// SIMATIC S7-200 SMART project (STEP 7-Micro/WIN SMART), CPU ST20

SYMBOL_TABLE 系统符号
Always_On        SM0.0    // 始终接通
First_Scan_On    SM0.1    // 仅在第一个扫描周期时接通
Clock_1s         SM0.5    // 针对 1 s 的周期时间，时钟脉冲接通 0.5 s，断开 0.5 s.
Time_0_Intrvl    SMB34    // 指定中断 0 的时间间隔（从 5 到 255，以 1 毫秒递增）。
END_SYMBOL_TABLE

ORGANIZATION_BLOCK MAIN:OB1
TITLE=程序注释
BEGIN
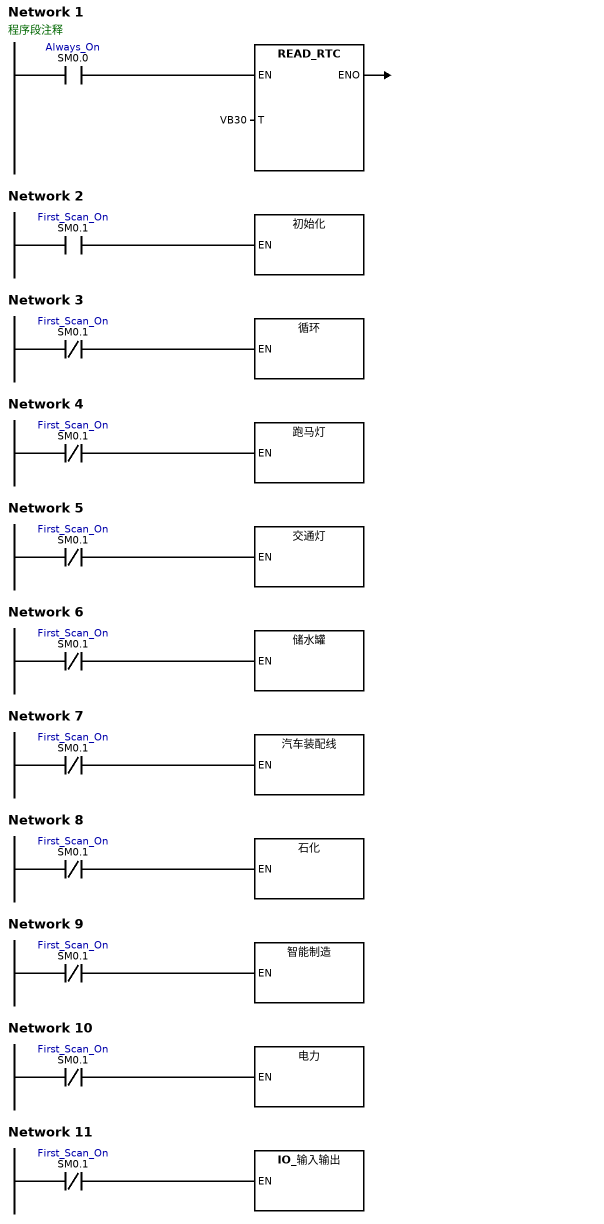
Network 1
// 程序段注释
LD     Always_On:SM0.0
TODR   VB30
Network 2
LD     First_Scan_On:SM0.1
CALL   初始化:SBR4
Network 3
LDN    First_Scan_On:SM0.1
CALL   循环:SBR14
Network 4
LDN    First_Scan_On:SM0.1
CALL   跑马灯:SBR0
Network 5
LDN    First_Scan_On:SM0.1
CALL   交通灯:SBR2
Network 6
// (network saved uncompiled; LAD cells follow)
// row 0: c0 -|/|- First_Scan_On:SM0.1  c1 --  c2 [储水罐 EN:=power@row0]
Network 7
LDN    First_Scan_On:SM0.1
CALL   汽车装配线:SBR7
Network 8
LDN    First_Scan_On:SM0.1
CALL   石化:SBR8
Network 9
LDN    First_Scan_On:SM0.1
CALL   智能制造:SBR9
Network 10
LDN    First_Scan_On:SM0.1
CALL   电力:SBR11
Network 11
LDN    First_Scan_On:SM0.1
CALL   IO_输入输出:SBR13
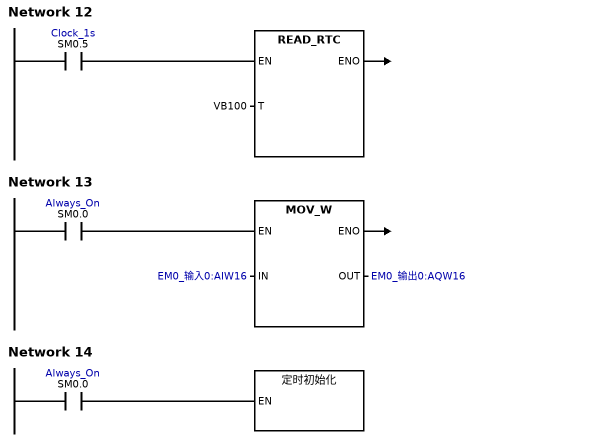
Network 12
LD     Clock_1s:SM0.5
TODR   VB100
Network 13
LD     Always_On:SM0.0
MOVW   EM0_输入0:AIW16, EM0_输出0:AQW16
Network 14
LD     Always_On:SM0.0
CALL   定时初始化:SBR1
END_ORGANIZATION_BLOCK

SUBROUTINE_BLOCK 跑马灯:SBR0
TITLE=子程序注释
BEGIN
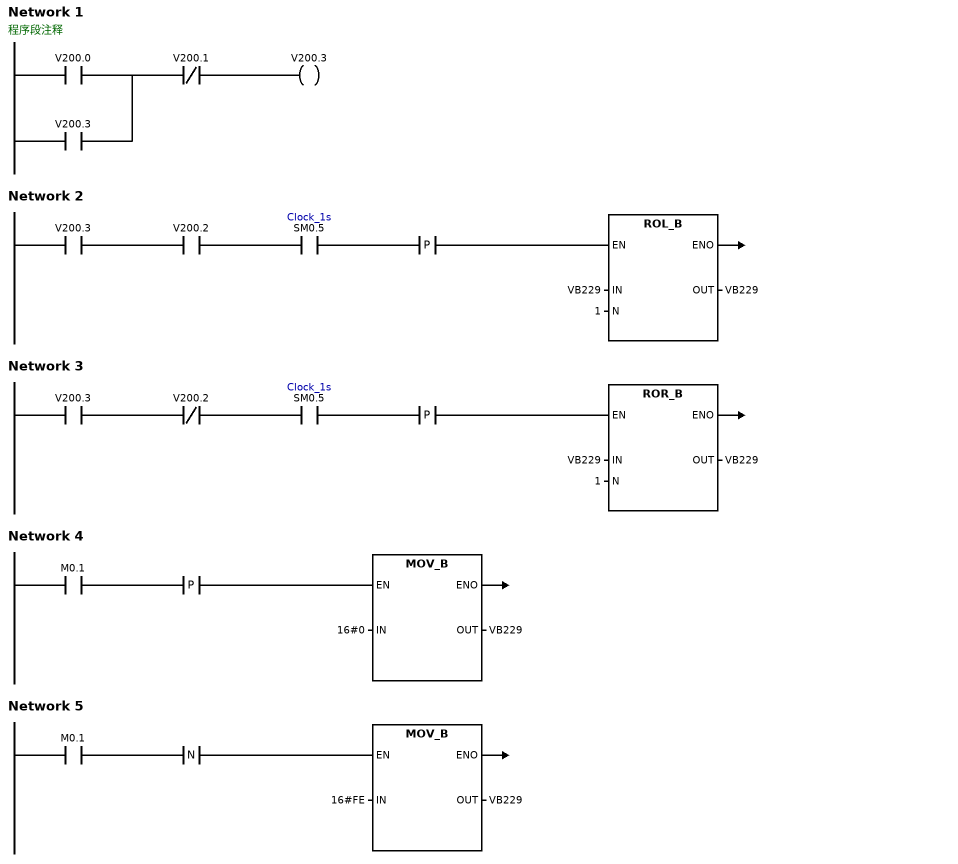
Network 1
// 程序段注释
LD     V200.0
O      V200.3
AN     V200.1
=      V200.3
Network 2
LD     V200.3
A      V200.2
A      Clock_1s:SM0.5
EU
RLB    VB229, 1
Network 3
LD     V200.3
AN     V200.2
A      Clock_1s:SM0.5
EU
RRB    VB229, 1
Network 4
LD     M0.1
EU
MOVB   16#0, VB229
Network 5
LD     M0.1
ED
MOVB   16#FE, VB229
END_SUBROUTINE_BLOCK

SUBROUTINE_BLOCK 定时初始化:SBR1
TITLE=
BEGIN
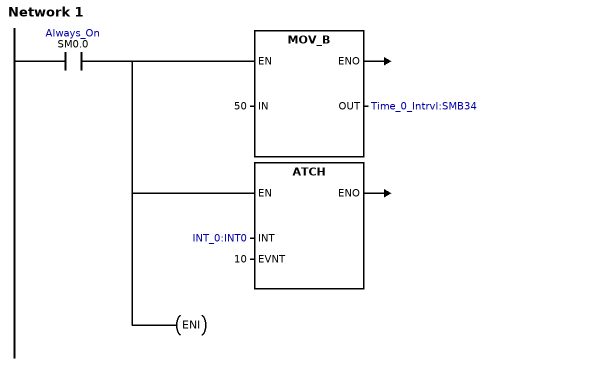
Network 1
LD     Always_On:SM0.0
MOVB   50, Time_0_Intrvl:SMB34
ATCH   INT_0:INT0, 10
ENI
END_SUBROUTINE_BLOCK

SUBROUTINE_BLOCK 交通灯:SBR2
TITLE=
BEGIN
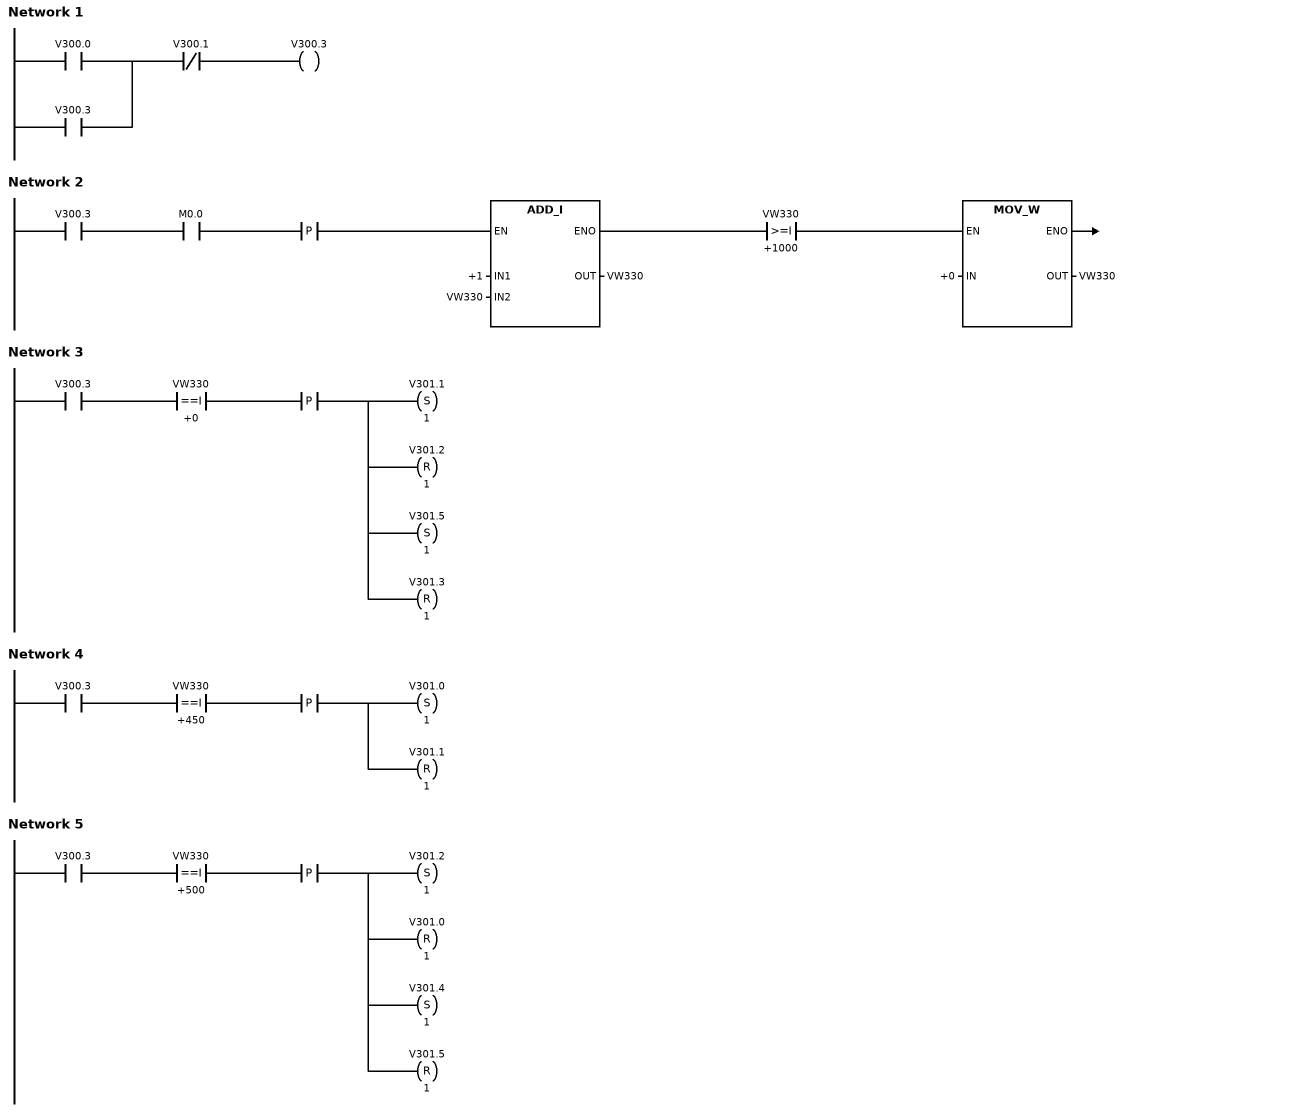
Network 1
LD     V300.0
O      V300.3
AN     V300.1
=      V300.3
Network 2
LD     V300.3
A      M0.0
EU
+I     +1, VW330
AENO
AW>=   VW330, +1000
MOVW   +0, VW330
Network 3
LD     V300.3
AW=    VW330, +0
EU
S      V301.1, 1
R      V301.2, 1
S      V301.5, 1
R      V301.3, 1
Network 4
LD     V300.3
AW=    VW330, +450
EU
S      V301.0, 1
R      V301.1, 1
Network 5
LD     V300.3
AW=    VW330, +500
EU
S      V301.2, 1
R      V301.0, 1
S      V301.4, 1
R      V301.5, 1
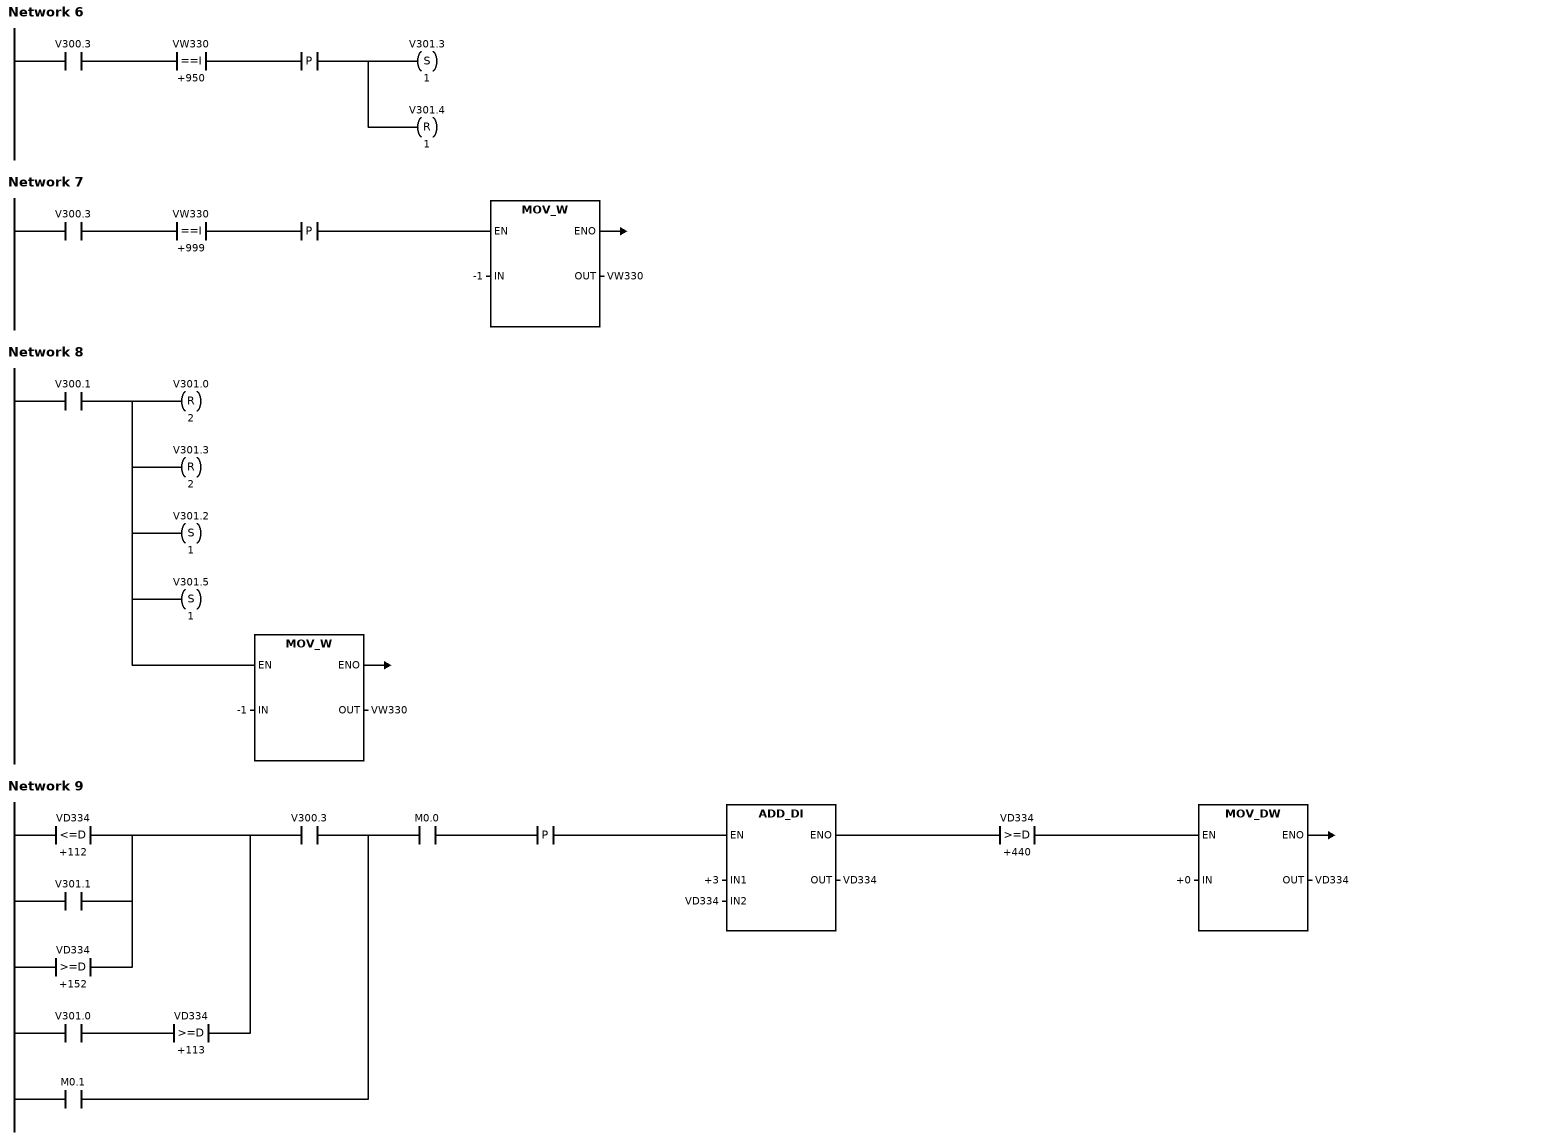
Network 6
LD     V300.3
AW=    VW330, +950
EU
S      V301.3, 1
R      V301.4, 1
Network 7
LD     V300.3
AW=    VW330, +999
EU
MOVW   -1, VW330
Network 8
LD     V300.1
R      V301.0, 2
R      V301.3, 2
S      V301.2, 1
S      V301.5, 1
MOVW   -1, VW330
Network 9
LDD<=  VD334, +112
O      V301.1
OD>=   VD334, +152
LD     V301.0
AD>=   VD334, +113
OLD
A      V300.3
O      M0.1
A      M0.0
EU
+D     +3, VD334
AENO
AD>=   VD334, +440
MOVD   +0, VD334
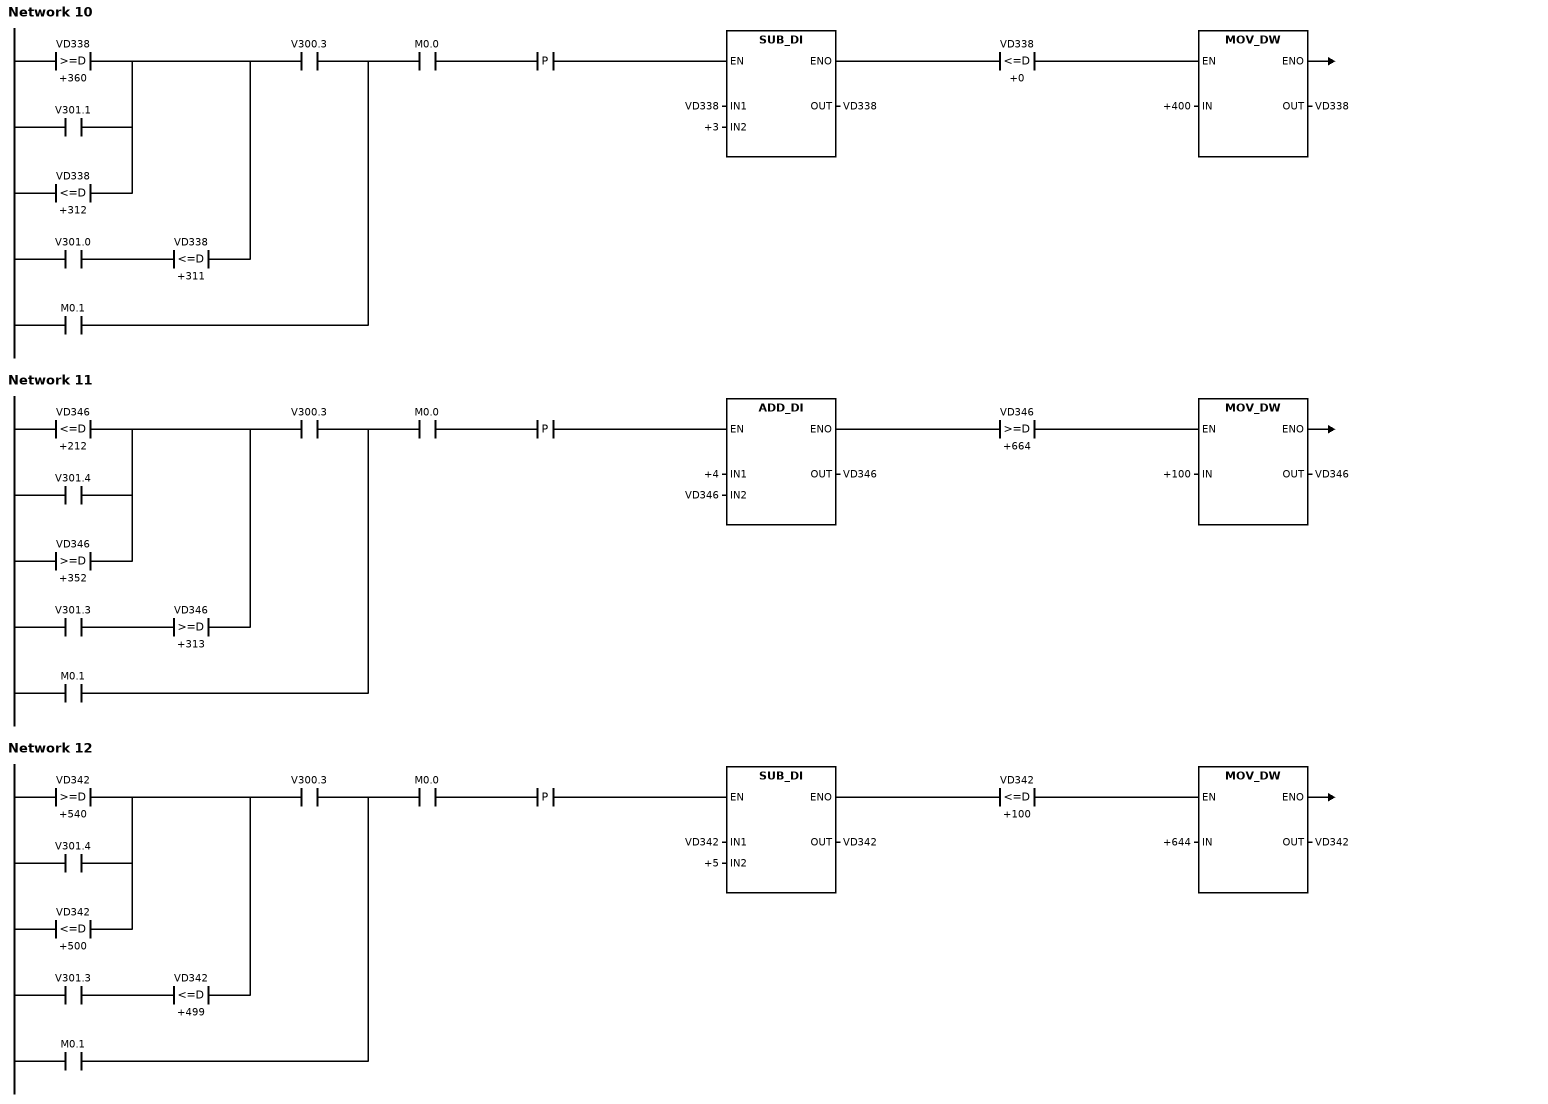
Network 10
LDD>=  VD338, +360
O      V301.1
OD<=   VD338, +312
LD     V301.0
AD<=   VD338, +311
OLD
A      V300.3
O      M0.1
A      M0.0
EU
-D     +3, VD338
AENO
AD<=   VD338, +0
MOVD   +400, VD338
Network 11
LDD<=  VD346, +212
O      V301.4
OD>=   VD346, +352
LD     V301.3
AD>=   VD346, +313
OLD
A      V300.3
O      M0.1
A      M0.0
EU
+D     +4, VD346
AENO
AD>=   VD346, +664
MOVD   +100, VD346
Network 12
LDD>=  VD342, +540
O      V301.4
OD<=   VD342, +500
LD     V301.3
AD<=   VD342, +499
OLD
A      V300.3
O      M0.1
A      M0.0
EU
-D     +5, VD342
AENO
AD<=   VD342, +100
MOVD   +644, VD342
END_SUBROUTINE_BLOCK

SUBROUTINE_BLOCK 模拟量输出:SBR3
TITLE=
VAR_INPUT
In_Data:REAL;	// LD0 
HH:REAL;	// LD4 
LL:REAL;	// LD8 
END_VAR
VAR_OUTPUT
AQW_:INT;	// LW12 
END_VAR
BEGIN
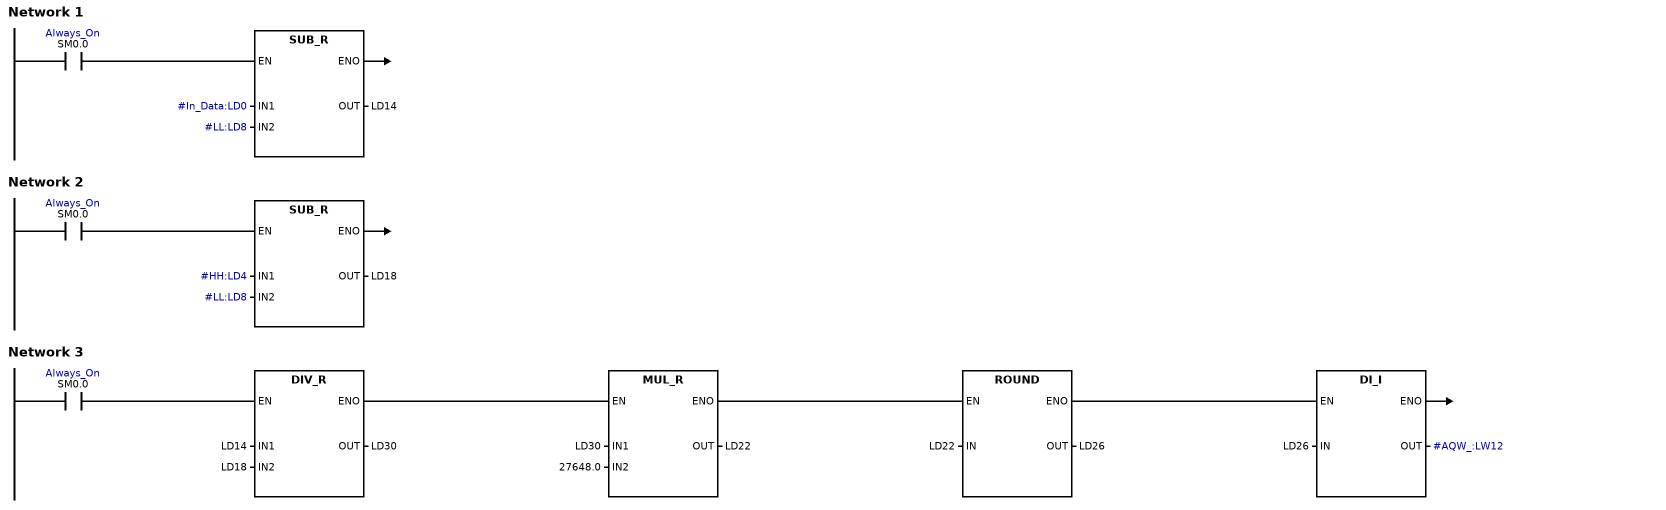
Network 1
LD     Always_On:SM0.0
MOVR   #In_Data:LD0, LD14
-R     #LL:LD8, LD14
Network 2
LD     Always_On:SM0.0
MOVR   #HH:LD4, LD18
-R     #LL:LD8, LD18
Network 3
LD     Always_On:SM0.0
MOVR   LD14, LD30
AENO
/R     LD18, LD30
AENO
MOVR   LD30, LD22
AENO
*R     27648.0, LD22
AENO
ROUND  LD22, LD26
AENO
DTI    LD26, #AQW_:LW12
END_SUBROUTINE_BLOCK

SUBROUTINE_BLOCK 初始化:SBR4
TITLE=
BEGIN
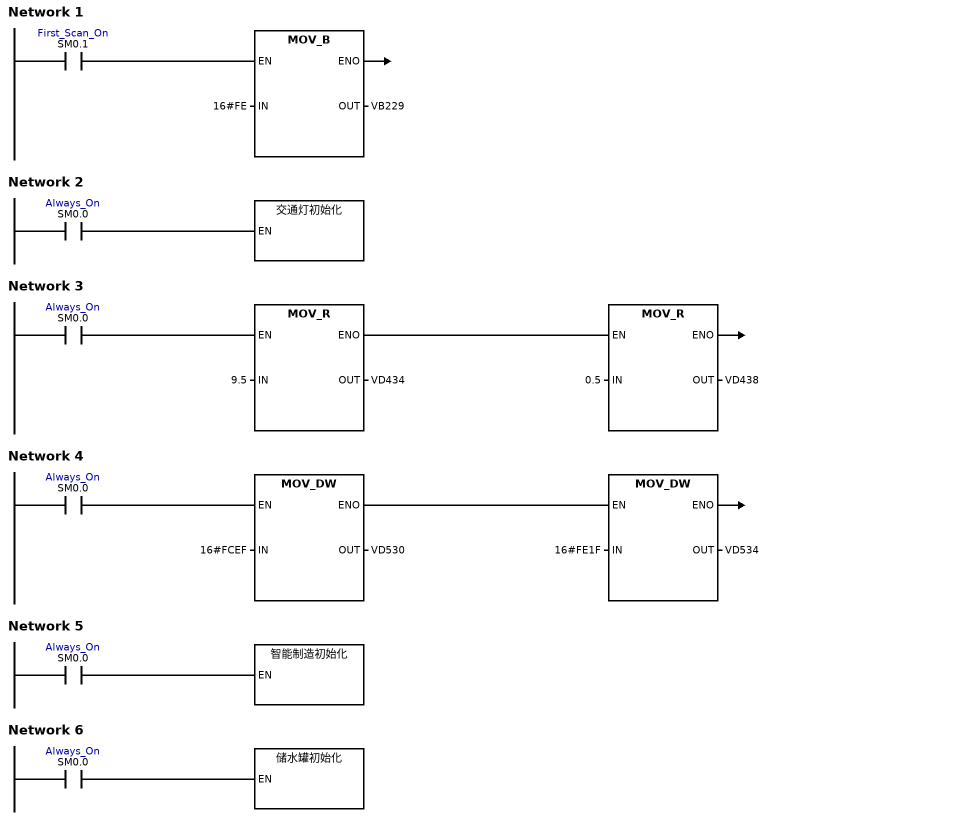
Network 1
LD     First_Scan_On:SM0.1
MOVB   16#FE, VB229
Network 2
LD     Always_On:SM0.0
CALL   交通灯初始化:SBR5
Network 3
LD     Always_On:SM0.0
MOVR   9.5, VD434
AENO
MOVR   0.5, VD438
Network 4
LD     Always_On:SM0.0
MOVD   16#FCEF, VD530
AENO
MOVD   16#FE1F, VD534
Network 5
LD     Always_On:SM0.0
CALL   智能制造初始化:SBR10
Network 6
LD     Always_On:SM0.0
CALL   储水罐初始化:SBR12
END_SUBROUTINE_BLOCK

SUBROUTINE_BLOCK 交通灯初始化:SBR5
TITLE=
BEGIN
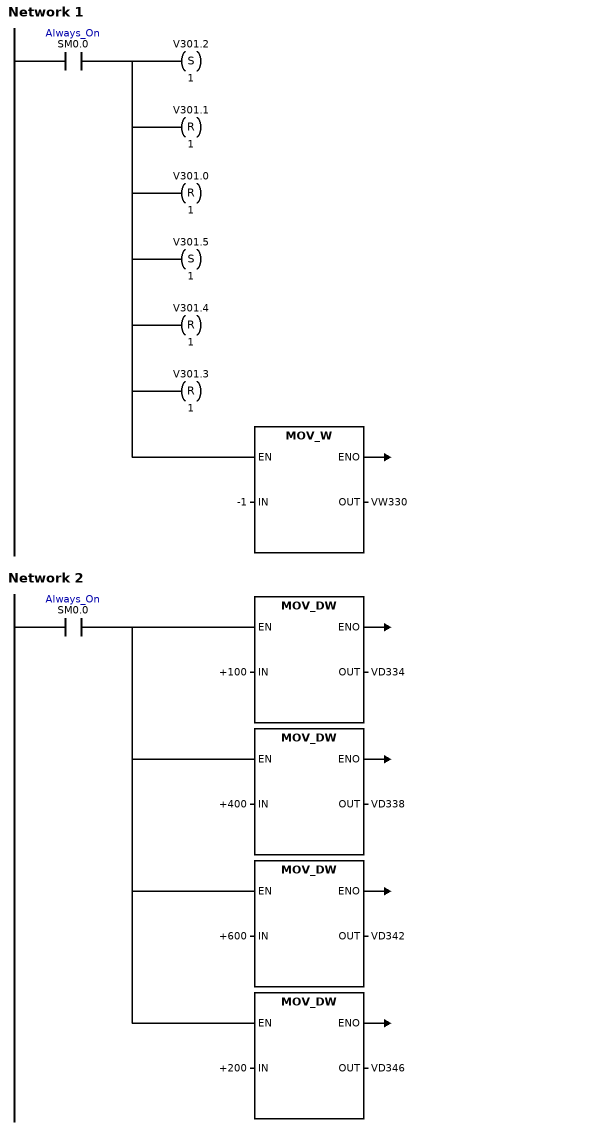
Network 1
LD     Always_On:SM0.0
S      V301.2, 1
R      V301.1, 1
R      V301.0, 1
S      V301.5, 1
R      V301.4, 1
R      V301.3, 1
MOVW   -1, VW330
Network 2
LD     Always_On:SM0.0
MOVD   +100, VD334
MOVD   +400, VD338
MOVD   +600, VD342
MOVD   +200, VD346
END_SUBROUTINE_BLOCK

SUBROUTINE_BLOCK 储水罐:SBR6
TITLE=
BEGIN
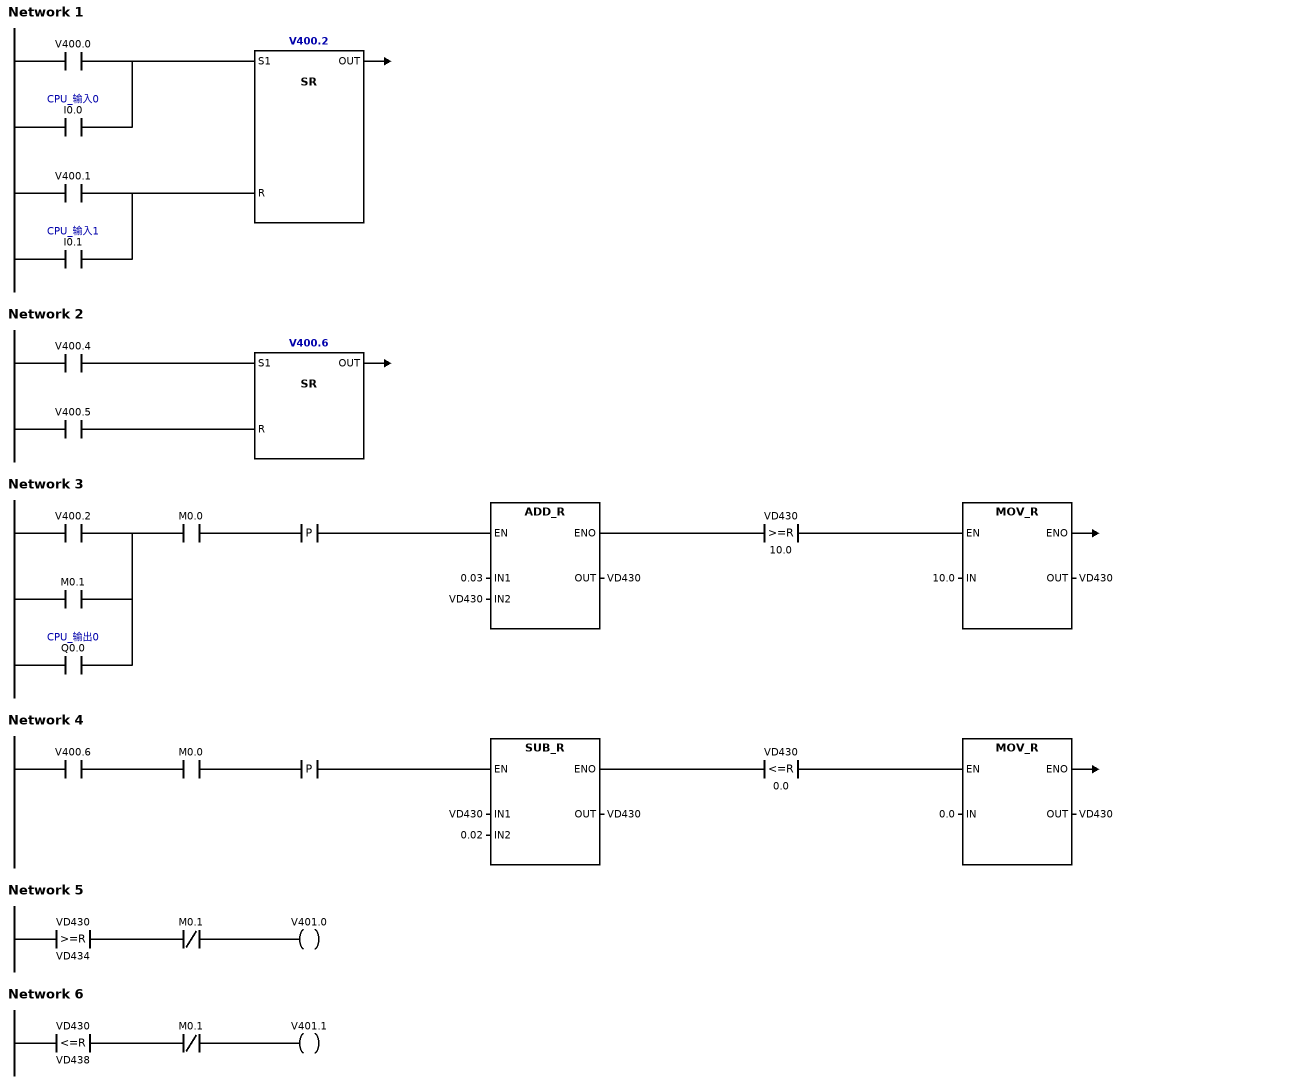
Network 1
LD     V400.0
O      CPU_输入0:I0.0
LD     V400.1
O      CPU_输入1:I0.1
NOT
A      V400.2
OLD
=      V400.2
Network 2
LD     V400.4
LD     V400.5
NOT
A      V400.6
OLD
=      V400.6
Network 3
LD     V400.2
O      M0.1
O      CPU_输出0:Q0.0
A      M0.0
EU
+R     0.03, VD430
AENO
AR>=   VD430, 10.0
MOVR   10.0, VD430
Network 4
LD     V400.6
A      M0.0
EU
-R     0.02, VD430
AENO
AR<=   VD430, 0.0
MOVR   0.0, VD430
Network 5
LDR>=  VD430, VD434
AN     M0.1
=      V401.0
Network 6
LDR<=  VD430, VD438
AN     M0.1
=      V401.1
END_SUBROUTINE_BLOCK

SUBROUTINE_BLOCK 汽车装配线:SBR7
TITLE=
BEGIN
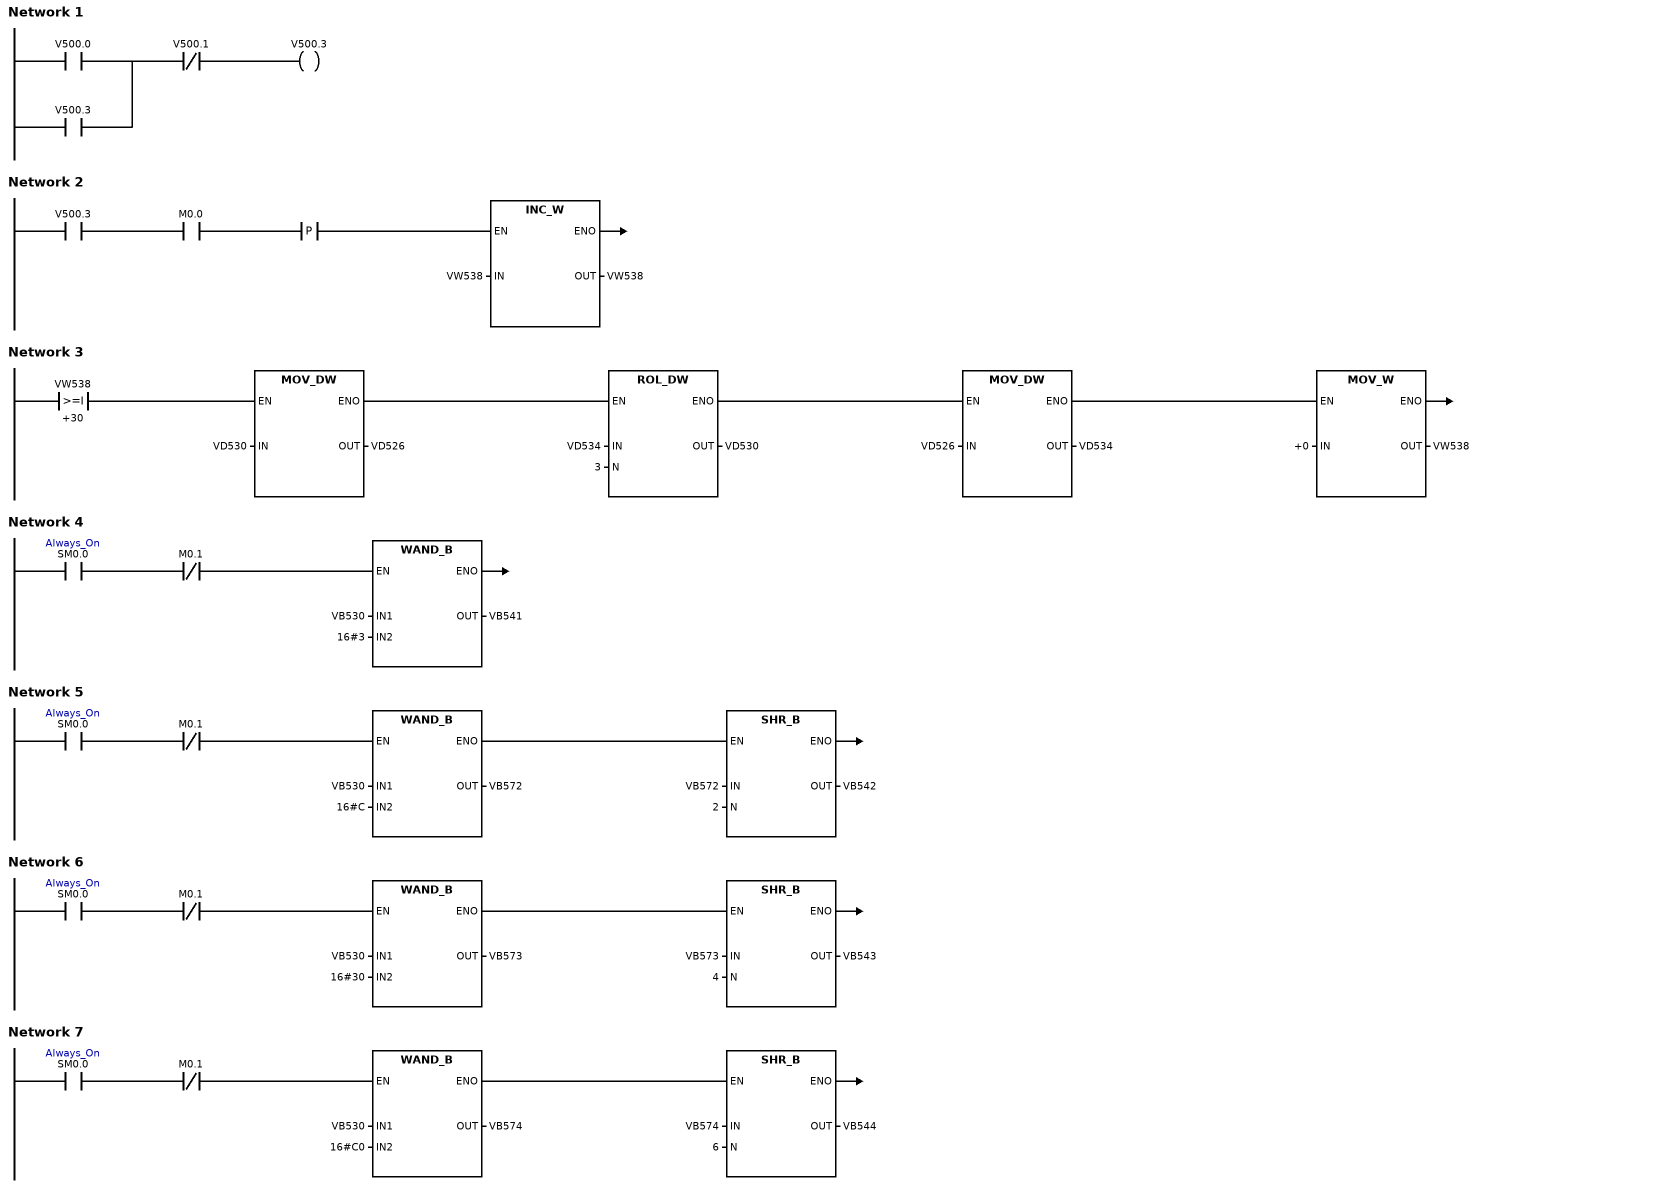
Network 1
LD     V500.0
O      V500.3
AN     V500.1
=      V500.3
Network 2
LD     V500.3
A      M0.0
EU
INCW   VW538
Network 3
LDW>=  VW538, +30
MOVD   VD530, VD526
AENO
MOVD   VD534, VD530
AENO
RLD    VD530, 3
AENO
MOVD   VD526, VD534
AENO
MOVW   +0, VW538
Network 4
LD     Always_On:SM0.0
AN     M0.1
MOVB   VB530, VB541
ANDB   16#3, VB541
Network 5
LD     Always_On:SM0.0
AN     M0.1
MOVB   VB530, VB572
AENO
ANDB   16#C, VB572
AENO
MOVB   VB572, VB542
SRB    VB542, 2
Network 6
LD     Always_On:SM0.0
AN     M0.1
MOVB   VB530, VB573
AENO
ANDB   16#30, VB573
AENO
MOVB   VB573, VB543
SRB    VB543, 4
Network 7
LD     Always_On:SM0.0
AN     M0.1
MOVB   VB530, VB574
AENO
ANDB   16#C0, VB574
AENO
MOVB   VB574, VB544
SRB    VB544, 6
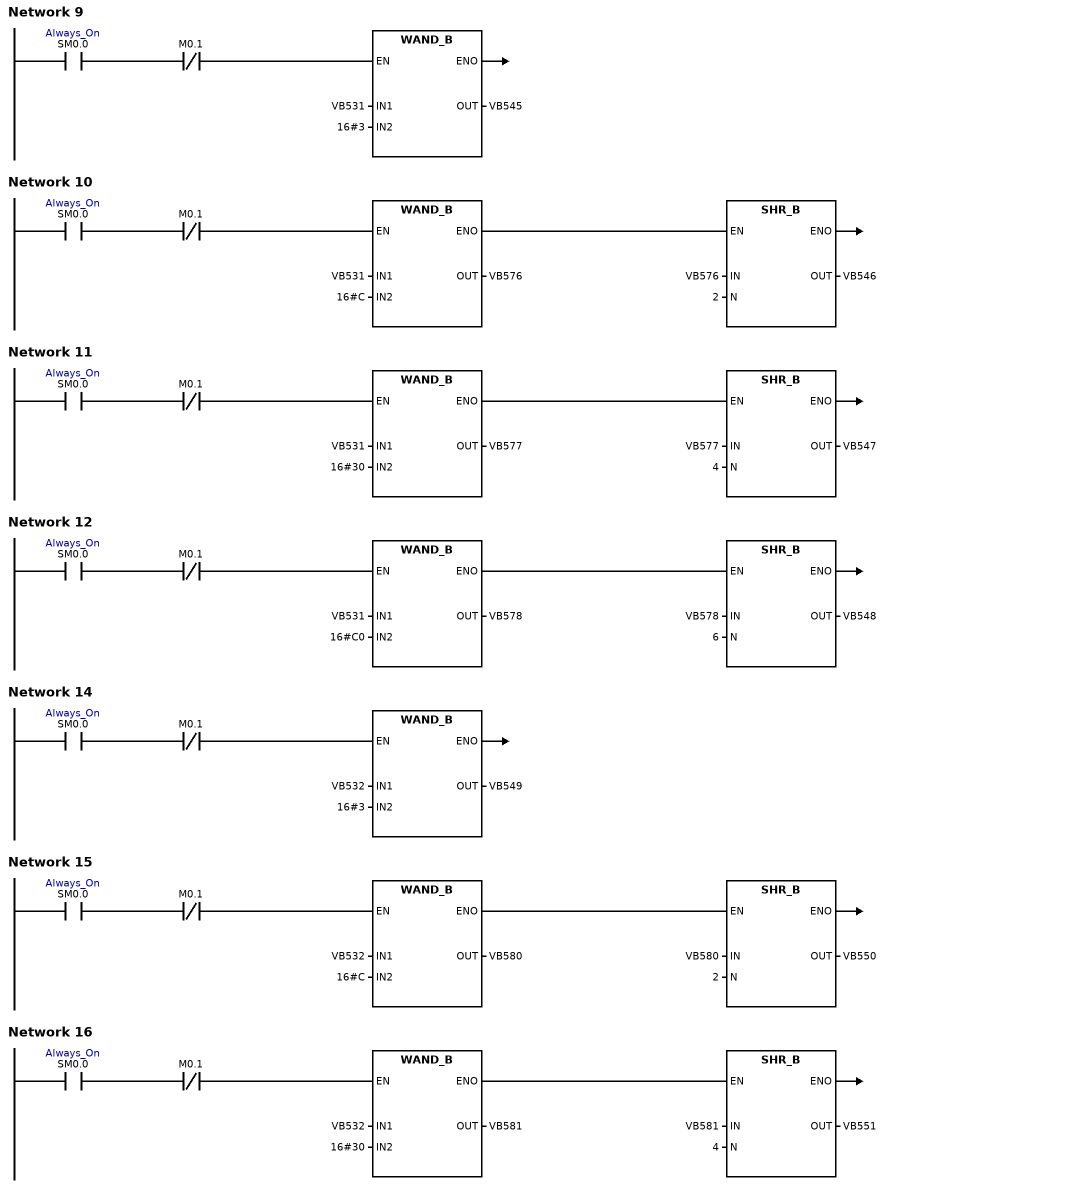
Network 9
LD     Always_On:SM0.0
AN     M0.1
MOVB   VB531, VB545
ANDB   16#3, VB545
Network 10
LD     Always_On:SM0.0
AN     M0.1
MOVB   VB531, VB576
AENO
ANDB   16#C, VB576
AENO
MOVB   VB576, VB546
SRB    VB546, 2
Network 11
LD     Always_On:SM0.0
AN     M0.1
MOVB   VB531, VB577
AENO
ANDB   16#30, VB577
AENO
MOVB   VB577, VB547
SRB    VB547, 4
Network 12
LD     Always_On:SM0.0
AN     M0.1
MOVB   VB531, VB578
AENO
ANDB   16#C0, VB578
AENO
MOVB   VB578, VB548
SRB    VB548, 6
Network 14
LD     Always_On:SM0.0
AN     M0.1
MOVB   VB532, VB549
ANDB   16#3, VB549
Network 15
LD     Always_On:SM0.0
AN     M0.1
MOVB   VB532, VB580
AENO
ANDB   16#C, VB580
AENO
MOVB   VB580, VB550
SRB    VB550, 2
Network 16
LD     Always_On:SM0.0
AN     M0.1
MOVB   VB532, VB581
AENO
ANDB   16#30, VB581
AENO
MOVB   VB581, VB551
SRB    VB551, 4
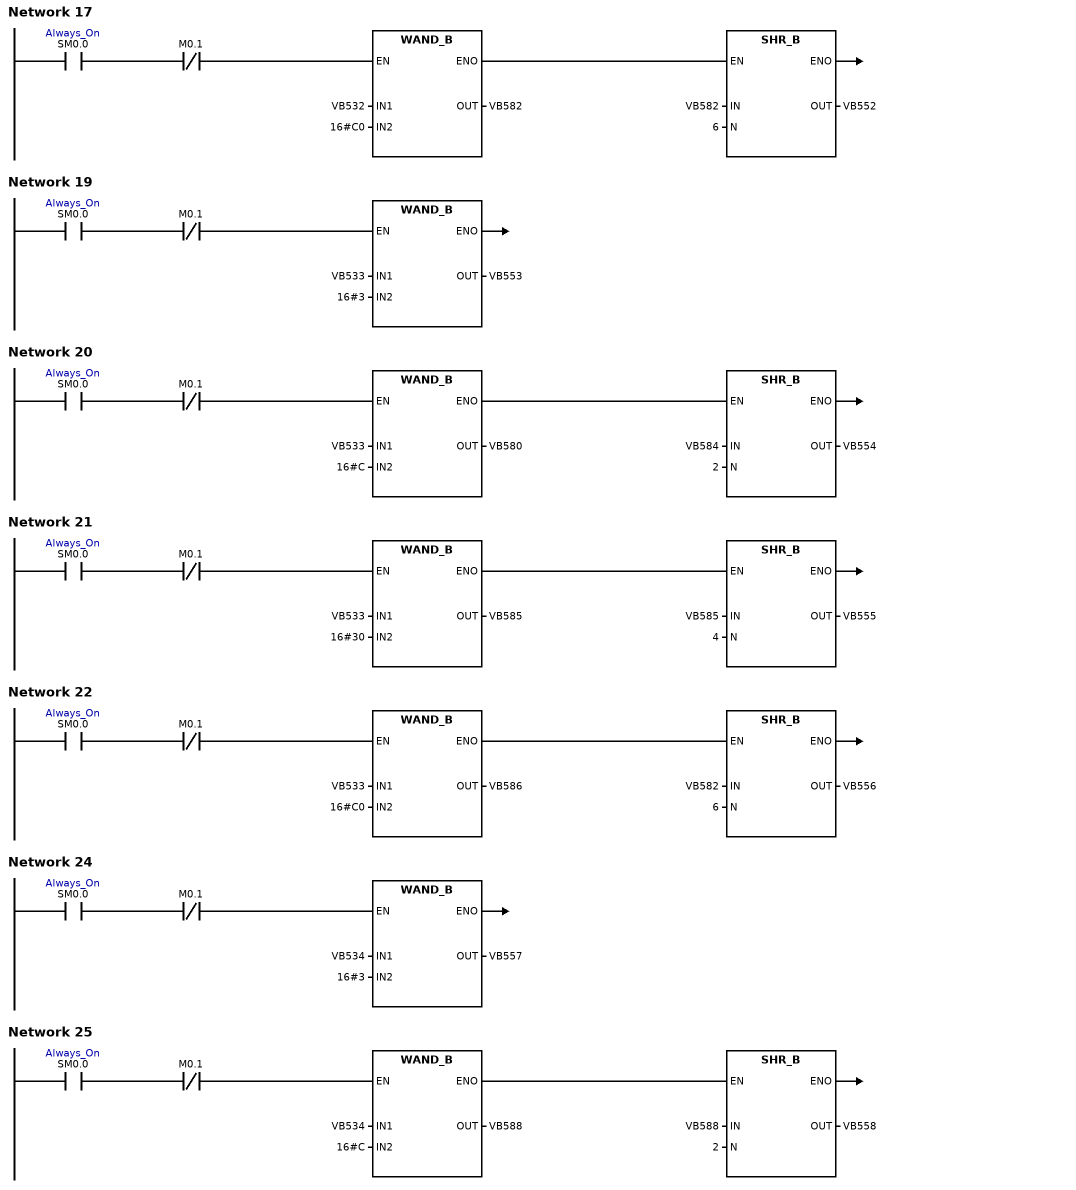
Network 17
LD     Always_On:SM0.0
AN     M0.1
MOVB   VB532, VB582
AENO
ANDB   16#C0, VB582
AENO
MOVB   VB582, VB552
SRB    VB552, 6
Network 19
LD     Always_On:SM0.0
AN     M0.1
MOVB   VB533, VB553
ANDB   16#3, VB553
Network 20
LD     Always_On:SM0.0
AN     M0.1
MOVB   VB533, VB580
AENO
ANDB   16#C, VB580
AENO
MOVB   VB584, VB554
SRB    VB554, 2
Network 21
LD     Always_On:SM0.0
AN     M0.1
MOVB   VB533, VB585
AENO
ANDB   16#30, VB585
AENO
MOVB   VB585, VB555
SRB    VB555, 4
Network 22
LD     Always_On:SM0.0
AN     M0.1
MOVB   VB533, VB586
AENO
ANDB   16#C0, VB586
AENO
MOVB   VB582, VB556
SRB    VB556, 6
Network 24
LD     Always_On:SM0.0
AN     M0.1
MOVB   VB534, VB557
ANDB   16#3, VB557
Network 25
LD     Always_On:SM0.0
AN     M0.1
MOVB   VB534, VB588
AENO
ANDB   16#C, VB588
AENO
MOVB   VB588, VB558
SRB    VB558, 2
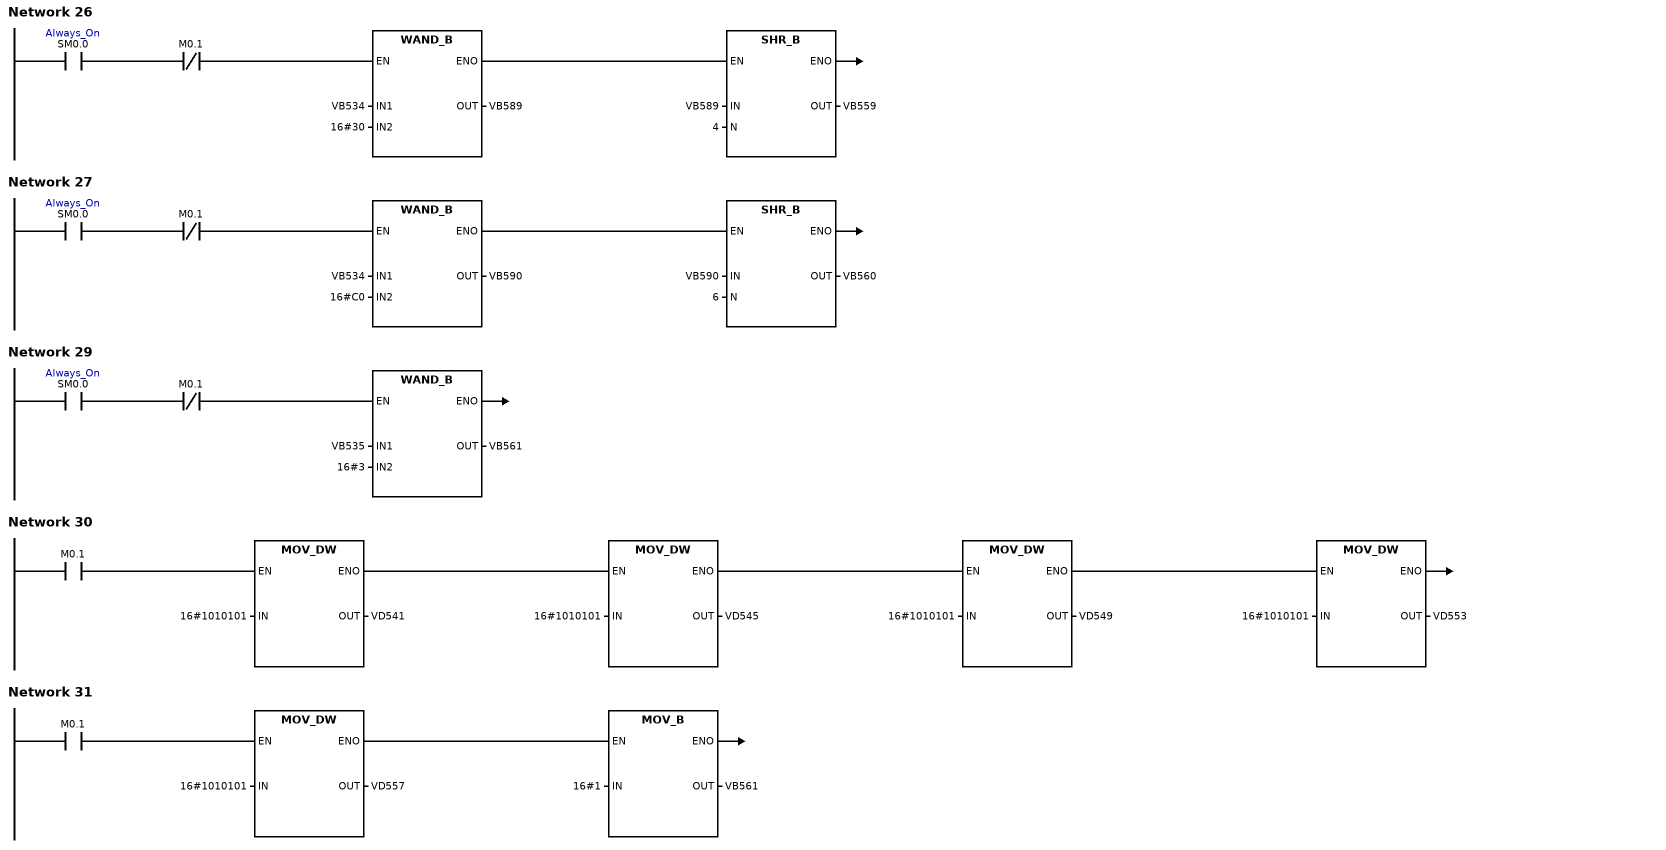
Network 26
LD     Always_On:SM0.0
AN     M0.1
MOVB   VB534, VB589
AENO
ANDB   16#30, VB589
AENO
MOVB   VB589, VB559
SRB    VB559, 4
Network 27
LD     Always_On:SM0.0
AN     M0.1
MOVB   VB534, VB590
AENO
ANDB   16#C0, VB590
AENO
MOVB   VB590, VB560
SRB    VB560, 6
Network 29
LD     Always_On:SM0.0
AN     M0.1
MOVB   VB535, VB561
ANDB   16#3, VB561
Network 30
LD     M0.1
MOVD   16#1010101, VD541
AENO
MOVD   16#1010101, VD545
AENO
MOVD   16#1010101, VD549
AENO
MOVD   16#1010101, VD553
Network 31
LD     M0.1
MOVD   16#1010101, VD557
AENO
MOVB   16#1, VB561
END_SUBROUTINE_BLOCK

SUBROUTINE_BLOCK 石化:SBR8
TITLE=
BEGIN
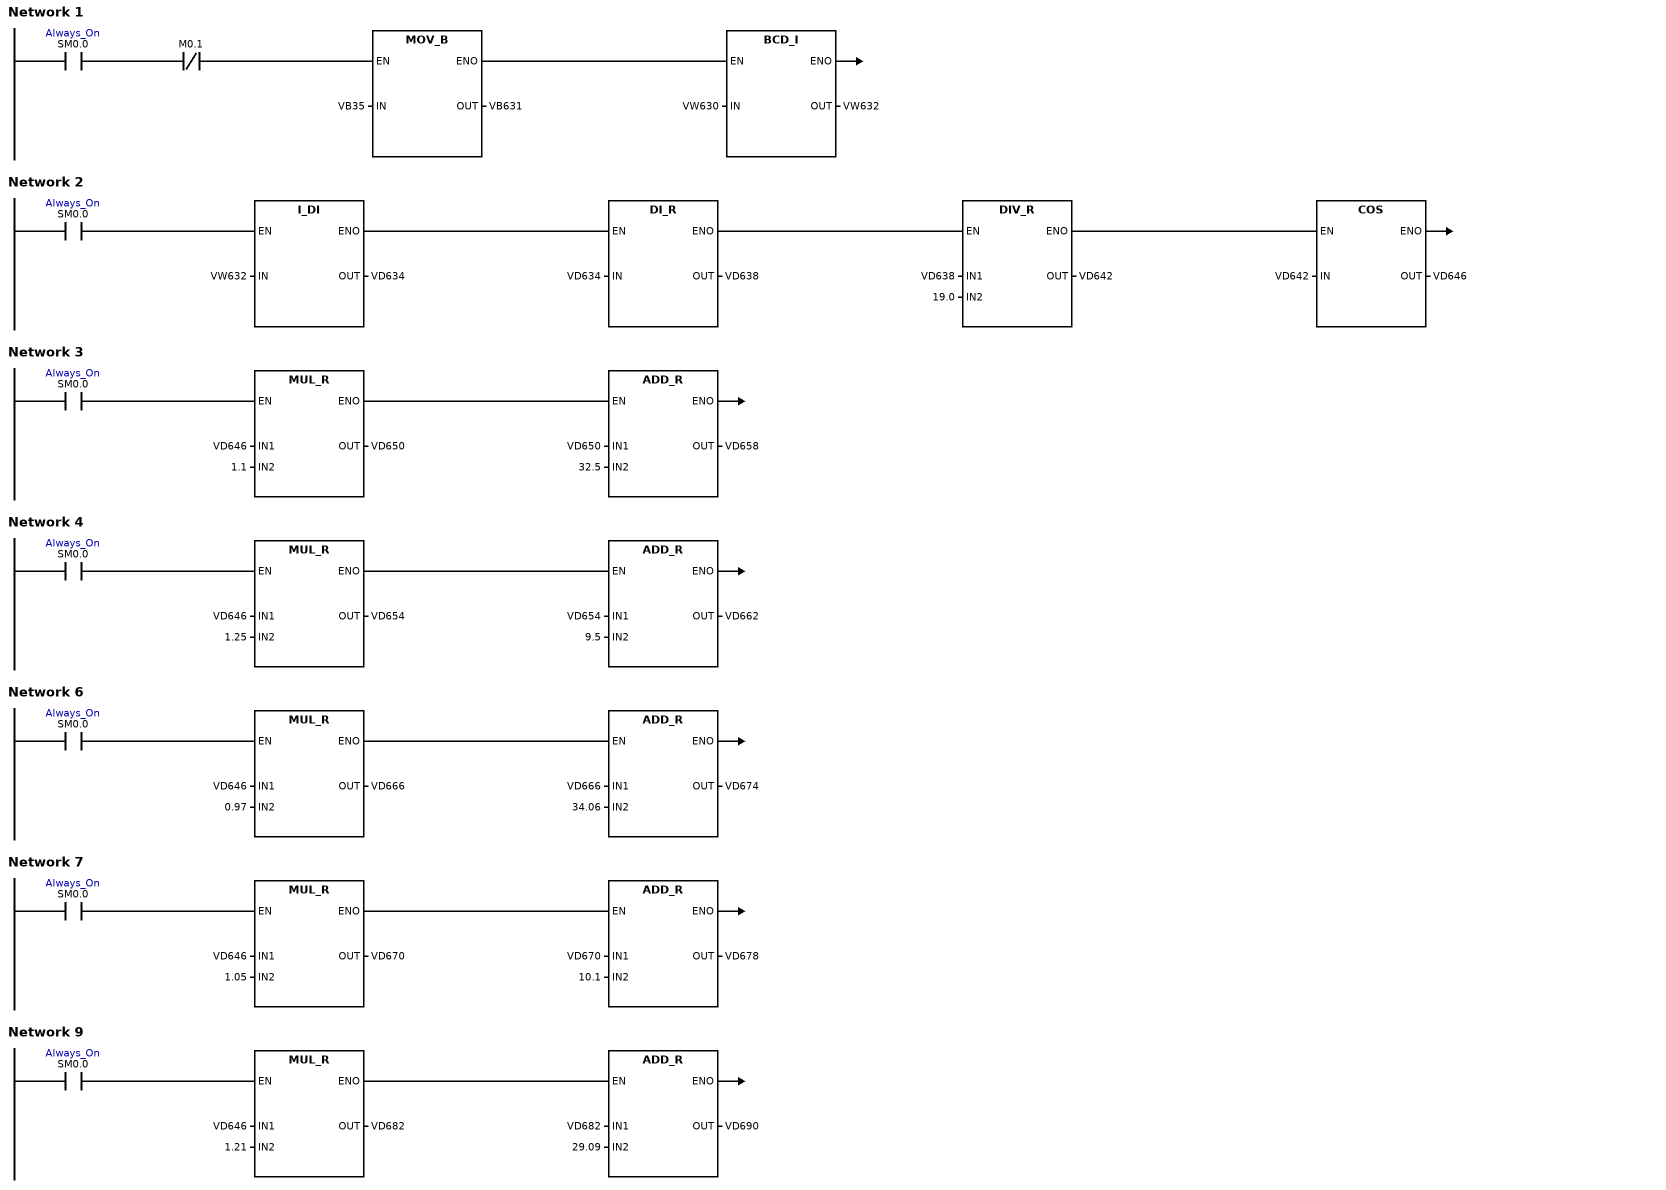
Network 1
LD     Always_On:SM0.0
AN     M0.1
MOVB   VB35, VB631
AENO
MOVW   VW630, VW632
BCDI   VW632
Network 2
LD     Always_On:SM0.0
ITD    VW632, VD634
AENO
DTR    VD634, VD638
AENO
MOVR   VD638, VD642
AENO
/R     19.0, VD642
AENO
COS    VD642, VD646
Network 3
LD     Always_On:SM0.0
MOVR   VD646, VD650
AENO
*R     1.1, VD650
AENO
MOVR   VD650, VD658
+R     32.5, VD658
Network 4
LD     Always_On:SM0.0
MOVR   VD646, VD654
AENO
*R     1.25, VD654
AENO
MOVR   VD654, VD662
+R     9.5, VD662
Network 6
LD     Always_On:SM0.0
MOVR   VD646, VD666
AENO
*R     0.97, VD666
AENO
MOVR   VD666, VD674
+R     34.06, VD674
Network 7
LD     Always_On:SM0.0
MOVR   VD646, VD670
AENO
*R     1.05, VD670
AENO
MOVR   VD670, VD678
+R     10.1, VD678
Network 9
LD     Always_On:SM0.0
MOVR   VD646, VD682
AENO
*R     1.21, VD682
AENO
MOVR   VD682, VD690
+R     29.09, VD690
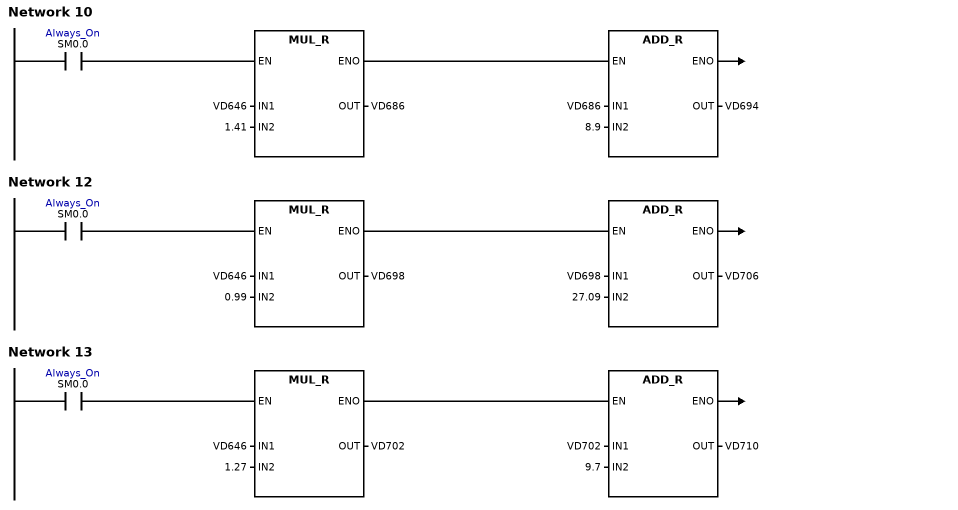
Network 10
LD     Always_On:SM0.0
MOVR   VD646, VD686
AENO
*R     1.41, VD686
AENO
MOVR   VD686, VD694
+R     8.9, VD694
Network 12
LD     Always_On:SM0.0
MOVR   VD646, VD698
AENO
*R     0.99, VD698
AENO
MOVR   VD698, VD706
+R     27.09, VD706
Network 13
LD     Always_On:SM0.0
MOVR   VD646, VD702
AENO
*R     1.27, VD702
AENO
MOVR   VD702, VD710
+R     9.7, VD710
END_SUBROUTINE_BLOCK

SUBROUTINE_BLOCK 智能制造:SBR9
TITLE=
BEGIN
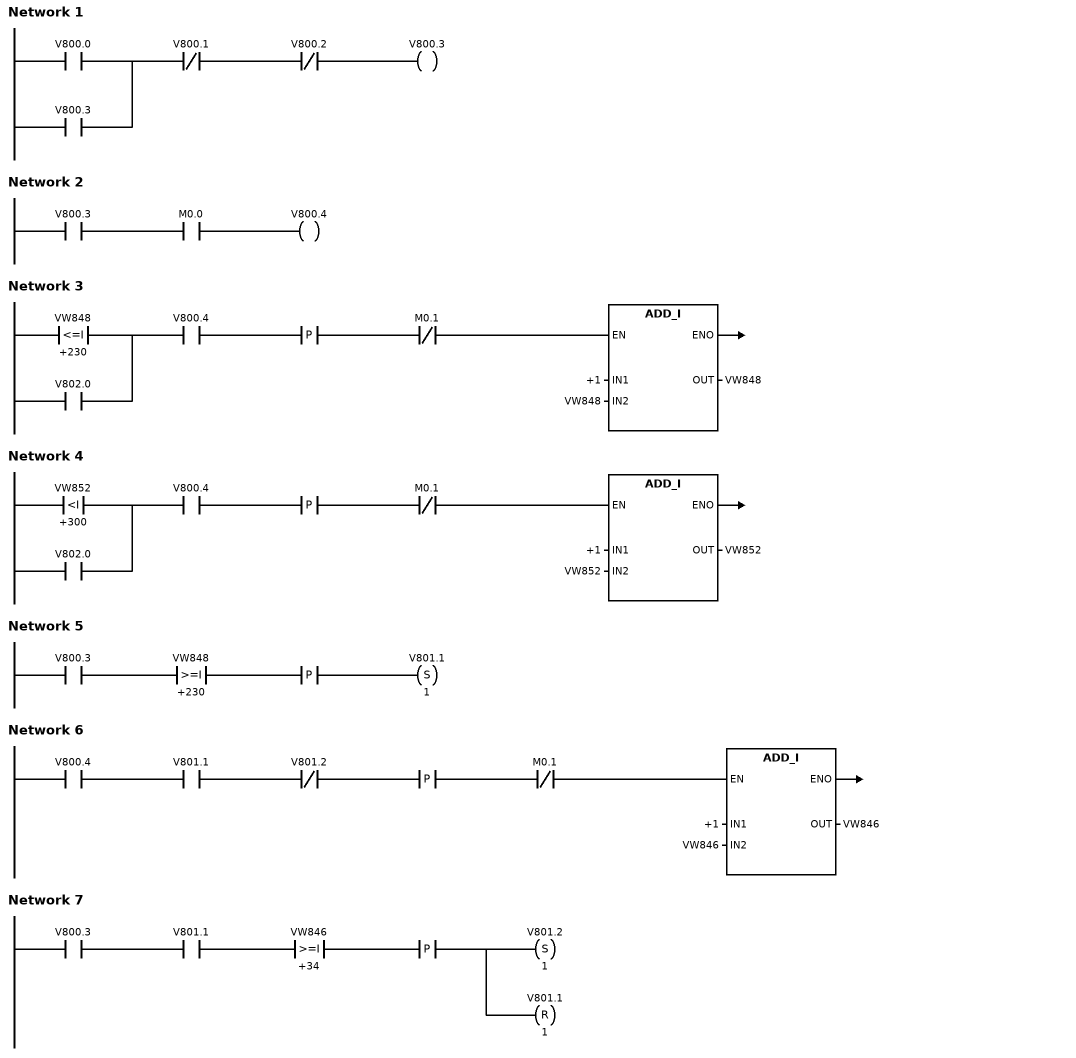
Network 1
LD     V800.0
O      V800.3
AN     V800.1
AN     V800.2
=      V800.3
Network 2
LD     V800.3
A      M0.0
=      V800.4
Network 3
LDW<=  VW848, +230
O      V802.0
A      V800.4
EU
AN     M0.1
+I     +1, VW848
Network 4
LDW<   VW852, +300
O      V802.0
A      V800.4
EU
AN     M0.1
+I     +1, VW852
Network 5
LD     V800.3
AW>=   VW848, +230
EU
S      V801.1, 1
Network 6
LD     V800.4
A      V801.1
AN     V801.2
EU
AN     M0.1
+I     +1, VW846
Network 7
LD     V800.3
A      V801.1
AW>=   VW846, +34
EU
S      V801.2, 1
R      V801.1, 1
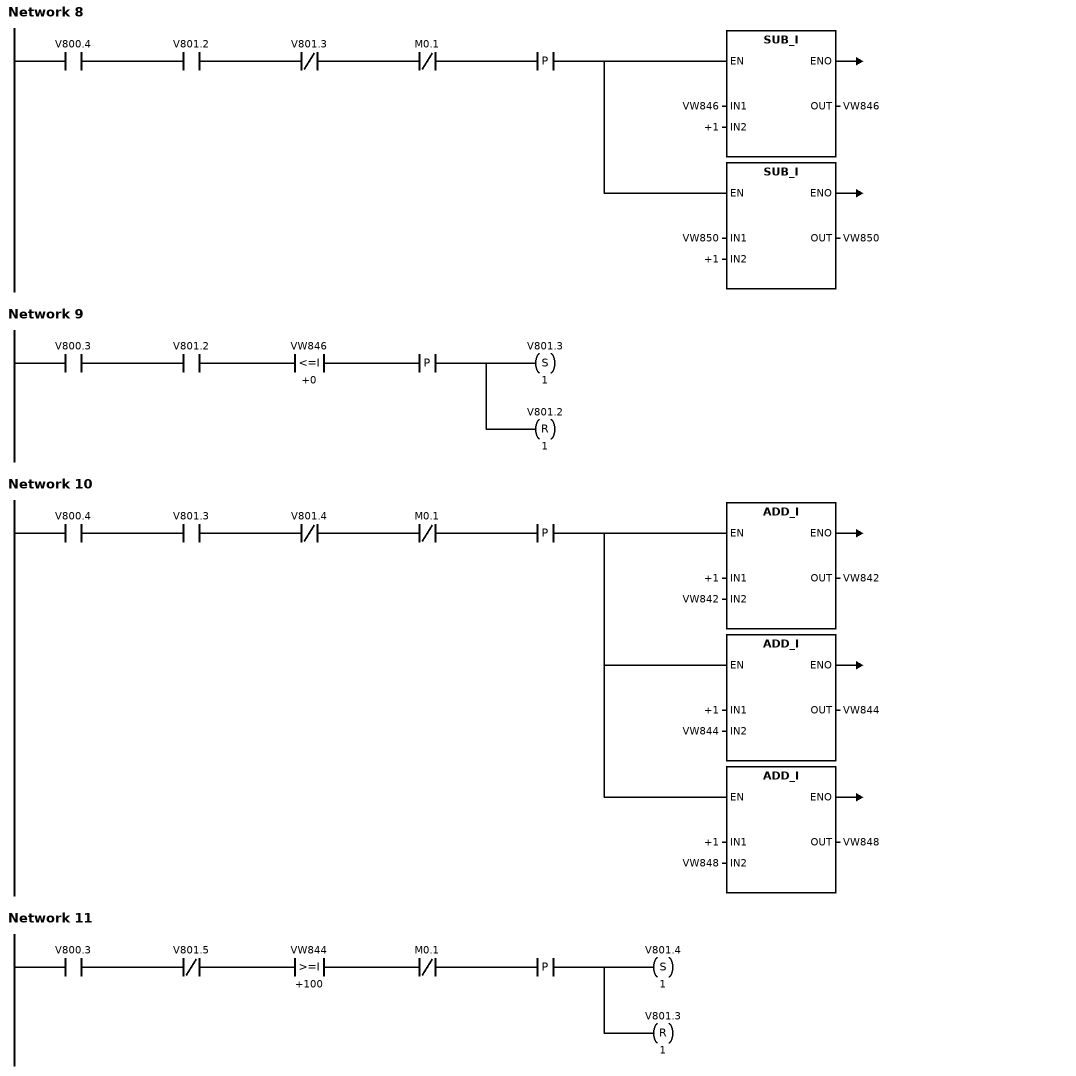
Network 8
LD     V800.4
A      V801.2
AN     V801.3
AN     M0.1
EU
-I     +1, VW846
-I     +1, VW850
Network 9
LD     V800.3
A      V801.2
AW<=   VW846, +0
EU
S      V801.3, 1
R      V801.2, 1
Network 10
LD     V800.4
A      V801.3
AN     V801.4
AN     M0.1
EU
+I     +1, VW842
+I     +1, VW844
+I     +1, VW848
Network 11
LD     V800.3
AN     V801.5
AW>=   VW844, +100
AN     M0.1
EU
S      V801.4, 1
R      V801.3, 1
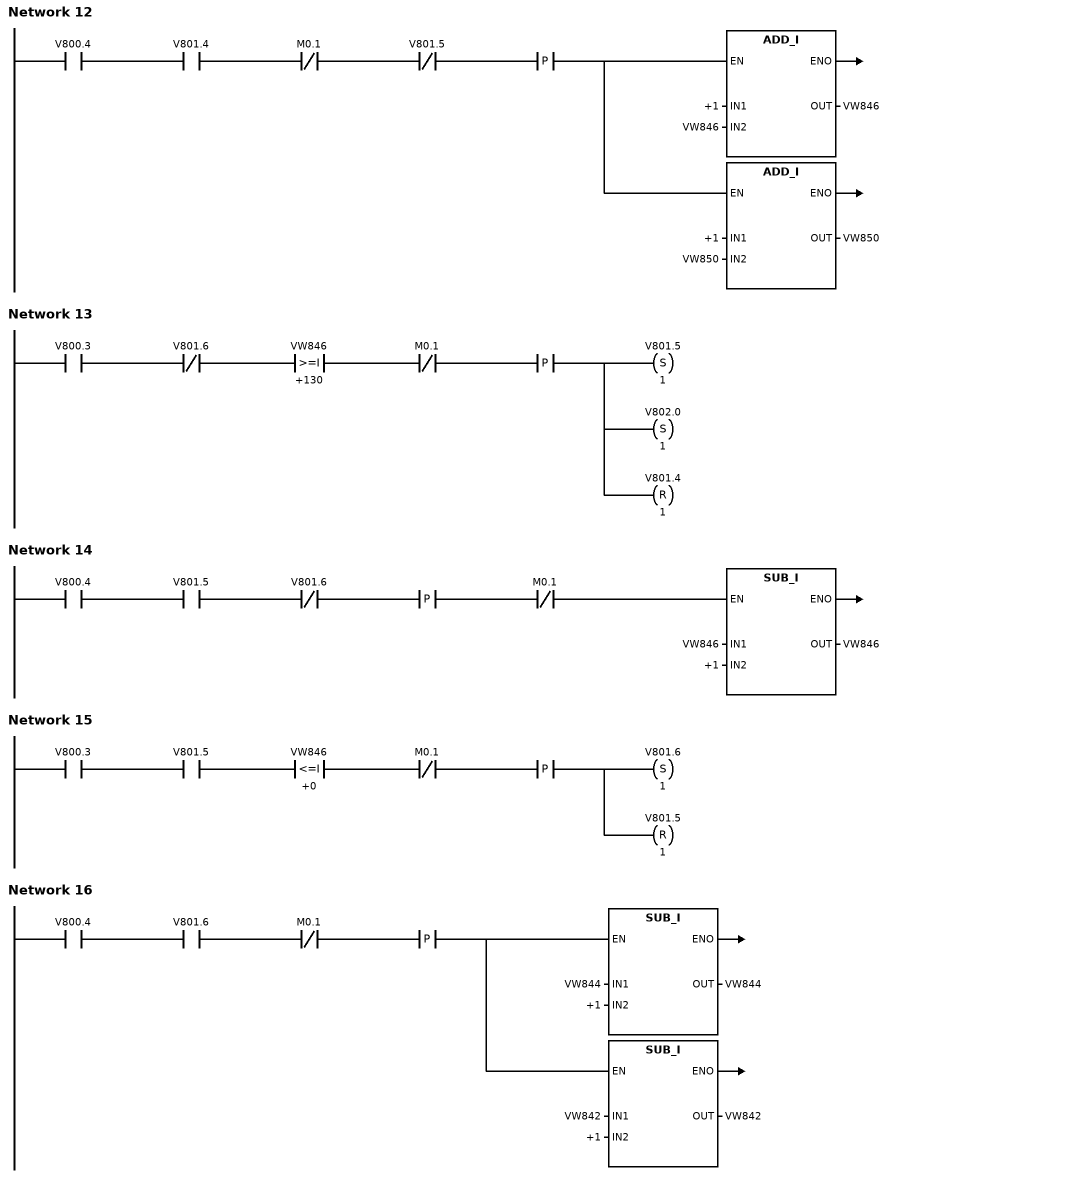
Network 12
LD     V800.4
A      V801.4
AN     M0.1
AN     V801.5
EU
+I     +1, VW846
+I     +1, VW850
Network 13
LD     V800.3
AN     V801.6
AW>=   VW846, +130
AN     M0.1
EU
S      V801.5, 1
S      V802.0, 1
R      V801.4, 1
Network 14
LD     V800.4
A      V801.5
AN     V801.6
EU
AN     M0.1
-I     +1, VW846
Network 15
LD     V800.3
A      V801.5
AW<=   VW846, +0
AN     M0.1
EU
S      V801.6, 1
R      V801.5, 1
Network 16
LD     V800.4
A      V801.6
AN     M0.1
EU
-I     +1, VW844
-I     +1, VW842
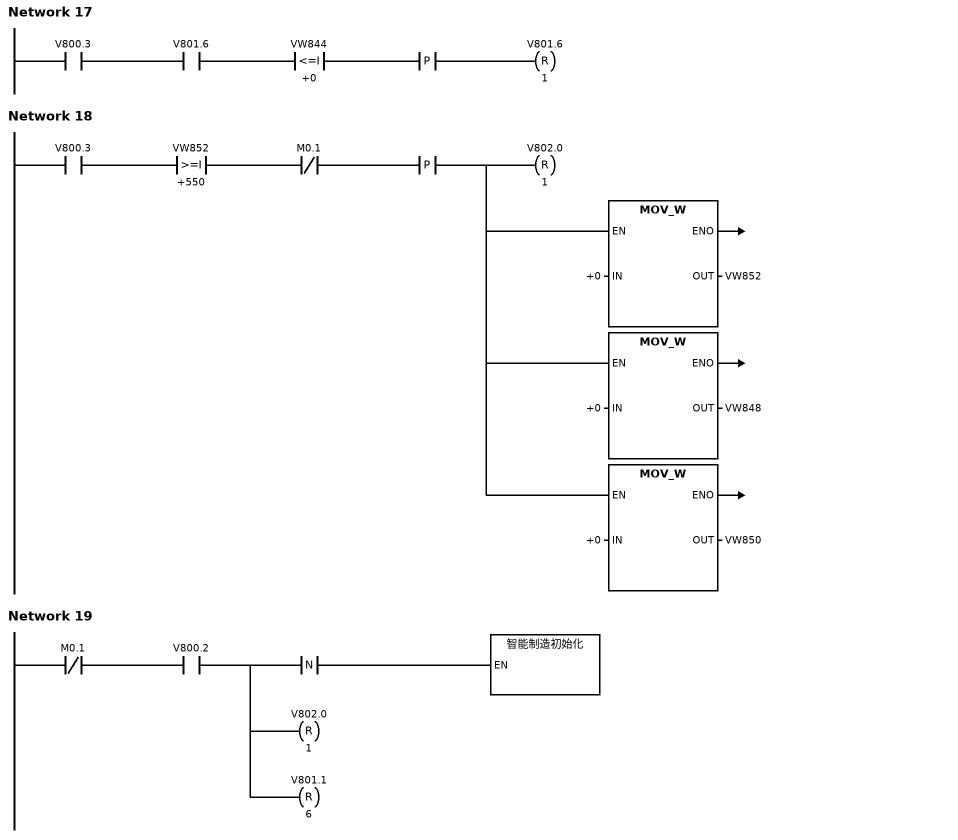
Network 17
LD     V800.3
A      V801.6
AW<=   VW844, +0
EU
R      V801.6, 1
Network 18
LD     V800.3
AW>=   VW852, +550
AN     M0.1
EU
R      V802.0, 1
MOVW   +0, VW852
MOVW   +0, VW848
MOVW   +0, VW850
Network 19
LDN    M0.1
A      V800.2
LPS
ED
CALL   智能制造初始化:SBR10
LRD
R      V802.0, 1
LPP
R      V801.1, 6
END_SUBROUTINE_BLOCK

SUBROUTINE_BLOCK 智能制造初始化:SBR10
TITLE=
BEGIN
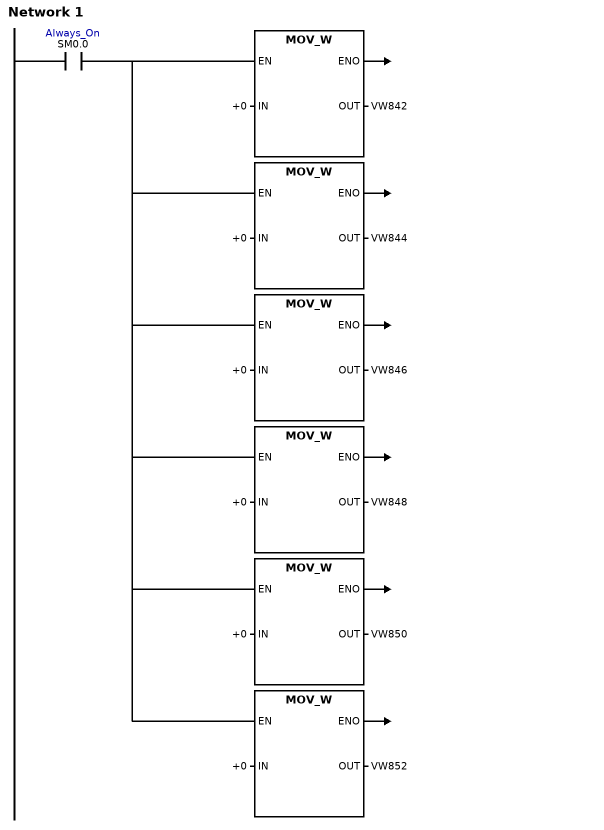
Network 1
LD     Always_On:SM0.0
MOVW   +0, VW842
MOVW   +0, VW844
MOVW   +0, VW846
MOVW   +0, VW848
MOVW   +0, VW850
MOVW   +0, VW852
END_SUBROUTINE_BLOCK

SUBROUTINE_BLOCK 电力:SBR11
TITLE=
BEGIN
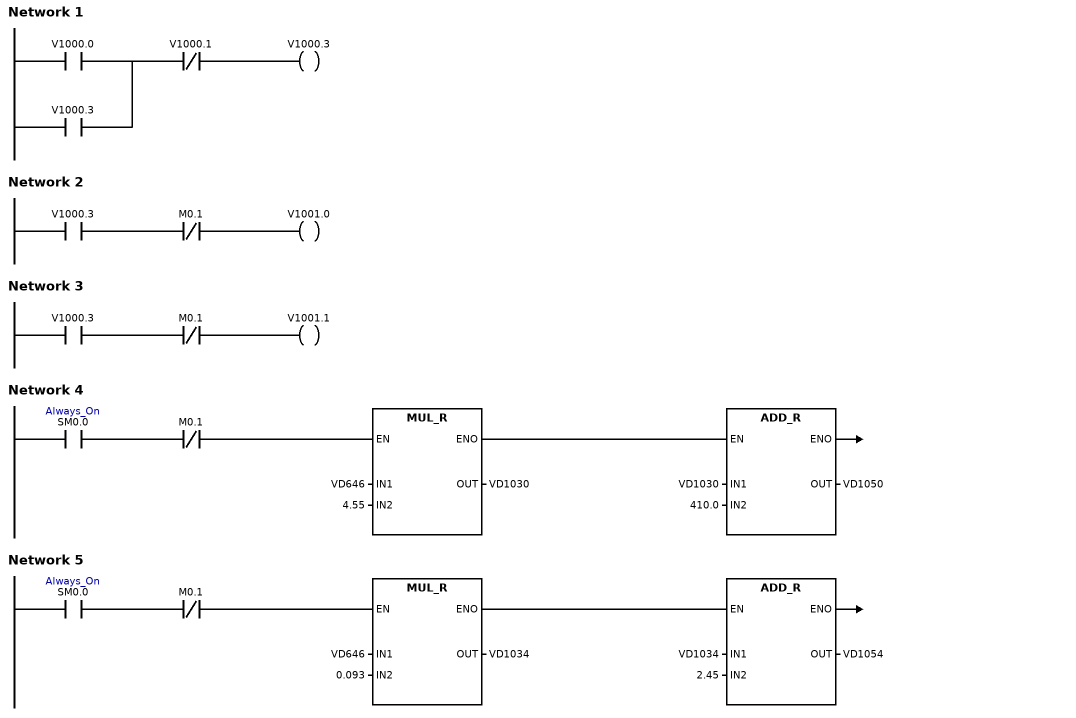
Network 1
LD     V1000.0
O      V1000.3
AN     V1000.1
=      V1000.3
Network 2
LD     V1000.3
AN     M0.1
=      V1001.0
Network 3
LD     V1000.3
AN     M0.1
=      V1001.1
Network 4
LD     Always_On:SM0.0
AN     M0.1
MOVR   VD646, VD1030
AENO
*R     4.55, VD1030
AENO
MOVR   VD1030, VD1050
+R     410.0, VD1050
Network 5
LD     Always_On:SM0.0
AN     M0.1
MOVR   VD646, VD1034
AENO
*R     0.093, VD1034
AENO
MOVR   VD1034, VD1054
+R     2.45, VD1054
END_SUBROUTINE_BLOCK

SUBROUTINE_BLOCK 储水罐初始化:SBR12
TITLE=
BEGIN
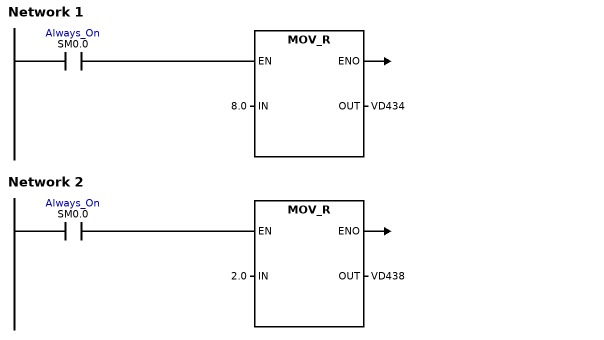
Network 1
LD     Always_On:SM0.0
MOVR   8.0, VD434
Network 2
LD     Always_On:SM0.0
MOVR   2.0, VD438
END_SUBROUTINE_BLOCK

SUBROUTINE_BLOCK IO_输入输出:SBR13
TITLE=
BEGIN
